// TIA Portal V16 export
// export: Created 2021-04-11T09:51:25.0986583Z, ExportSetting WithDefaults, DisplayName Totally Integrated Automation Portal, DisplayVersion V16, DisplayName TIA Portal Version Control Interface, DisplayVersion V16, DisplayName TIA Portal Openness, DisplayVersion V16, DisplayName STEP 7 Professional, DisplayVersion V16, DisplayName STEP 7 Safety, DisplayVersion V16, DisplayName WinCC Unified SCADA Engineering System, DisplayVersion V16
FUNCTION "preWorkBlock" : Void   // FC9, LAD
TITLE = Блок предработы
{ S7_Optimized_Access := 'TRUE' }
VERSION : 0.1
// Блок в котором организована работа цепей управления, аварийного останова и режимов работы
// stored: AutoNumber false, IsIECCheckEnabled false, SetENOAutomatically false, UDAEnableTagReadback false
BEGIN

REGION Network 1: удержание кнопки включение цепей управления
   // если аварийная кнопка не нажата то держим 2 секунды и цепи управления включаются
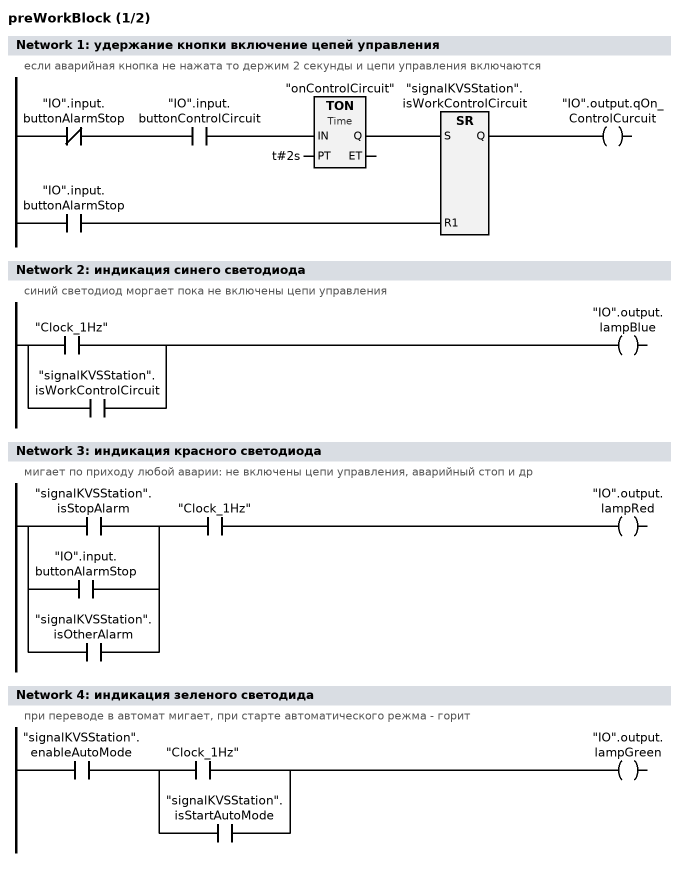
   RUNG wire#powerrail
      I_Contact( "IO".input.buttonAlarmStop )
      Contact( "IO".input.buttonControlCircuit )
      { S7_Templates := "time_type := Time" } "onControlCircuit".TON(pt := t#2s, et =>)
      S_SR(operand := "signalKVSStation".isWorkControlCircuit, r1 := wire#w1)
      Coil( "IO".output.qOn_ControlCurcuit )
   END_RUNG
   RUNG wire#powerrail
      Contact( "IO".input.buttonAlarmStop )
   END_RUNG wire#w1
   // the same network as SCL:
   "onControlCircuit".TON(IN := NOT "IO".input.buttonAlarmStop AND "IO".input.buttonControlCircuit, PT := t#2s);
   IF "onControlCircuit".Q THEN
       "signalKVSStation".isWorkControlCircuit := TRUE;   // SR flip-flop
   END_IF;
   IF "IO".input.buttonAlarmStop THEN "signalKVSStation".isWorkControlCircuit := FALSE; END_IF;
   "IO".output.qOn_ControlCurcuit := "signalKVSStation".isWorkControlCircuit;
END_REGION

REGION Network 2: индикация синего светодиода
   // синий светодиод моргает пока не включены цепи управления
   RUNG wire#powerrail
      Contact( "Clock_1Hz" )
      wire#w1
      Coil( "IO".output.lampBlue )
   END_RUNG
   RUNG wire#powerrail
      Contact( "signalKVSStation".isWorkControlCircuit )
   END_RUNG wire#w1
   // the same network as SCL:
   "IO".output.lampBlue := "Clock_1Hz" OR "signalKVSStation".isWorkControlCircuit;
END_REGION

REGION Network 3: индикация красного светодиода
   // мигает по приходу любой аварии: не включены цепи управления, аварийный стоп и др
   RUNG wire#powerrail
      Contact( "signalKVSStation".isStopAlarm )
      wire#w1
      Contact( "Clock_1Hz" )
      Coil( "IO".output.lampRed )
   END_RUNG
   RUNG wire#powerrail
      Contact( "IO".input.buttonAlarmStop )
   END_RUNG wire#w1
   RUNG wire#powerrail
      Contact( "signalKVSStation".isOtherAlarm )
   END_RUNG wire#w1
   // the same network as SCL:
   "IO".output.lampRed := ("signalKVSStation".isStopAlarm OR "IO".input.buttonAlarmStop OR "signalKVSStation".isOtherAlarm) AND "Clock_1Hz";
END_REGION

REGION Network 4: индикация зеленого светодида
   // при переводе в автомат мигает, при старте автоматического режма - горит
   RUNG wire#powerrail
      Contact( "signalKVSStation".enableAutoMode )
      wire#w1
      Contact( "Clock_1Hz" )
      wire#w2
      Coil( "IO".output.lampGreen )
   END_RUNG
   RUNG wire#w1
      Contact( "signalKVSStation".isStartAutoMode )
   END_RUNG wire#w2
   // the same network as SCL:
   "IO".output.lampGreen := "signalKVSStation".enableAutoMode AND ("Clock_1Hz" OR "signalKVSStation".isStartAutoMode);
END_REGION

REGION Network 5: разрешение на перевод в автоматический режим
   // при отсутствии аварий и нажатии кнопки автотоматического режима на панели. Данный сигнал используется как обратная связь по автоматическому и ручному режиму
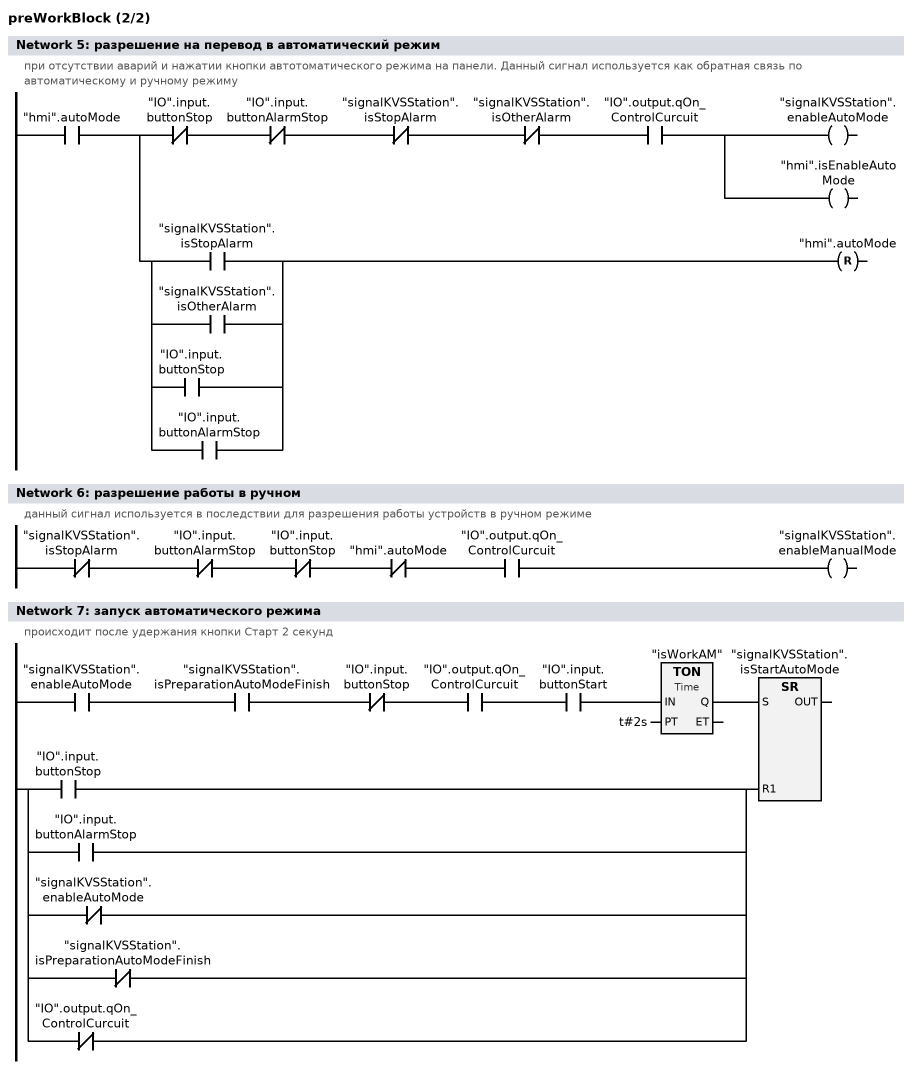
   RUNG wire#powerrail
      Contact( "hmi".autoMode )
      wire#w1
      I_Contact( "IO".input.buttonStop )
      I_Contact( "IO".input.buttonAlarmStop )
      I_Contact( "signalKVSStation".isStopAlarm )
      I_Contact( "signalKVSStation".isOtherAlarm )
      Contact( "IO".output.qOn_ControlCurcuit )
      wire#w2
      Coil( "signalKVSStation".enableAutoMode )
   END_RUNG
   RUNG wire#w2
      Coil( "hmi".isEnableAutoMode )
   END_RUNG
   RUNG wire#w1
      Contact( "signalKVSStation".isStopAlarm )
      wire#w3
      R_Coil( "hmi".autoMode )
   END_RUNG
   RUNG wire#w1
      Contact( "signalKVSStation".isOtherAlarm )
   END_RUNG wire#w3
   RUNG wire#w1
      Contact( "IO".input.buttonStop )
   END_RUNG wire#w3
   RUNG wire#w1
      Contact( "IO".input.buttonAlarmStop )
   END_RUNG wire#w3
   // the same network as SCL:
   "signalKVSStation".enableAutoMode := "hmi".autoMode AND NOT "IO".input.buttonStop AND NOT "IO".input.buttonAlarmStop AND NOT "signalKVSStation".isStopAlarm AND NOT "signalKVSStation".isOtherAlarm AND "IO".output.qOn_ControlCurcuit;
   "hmi".isEnableAutoMode := "signalKVSStation".enableAutoMode;
   IF "hmi".autoMode AND ("signalKVSStation".isStopAlarm OR "signalKVSStation".isOtherAlarm OR "IO".input.buttonStop OR "IO".input.buttonAlarmStop) THEN
       "hmi".autoMode := FALSE;
   END_IF;
END_REGION

REGION Network 6: разрешение работы в ручном
   // данный сигнал используется в последствии для разрешения работы устройств в ручном режиме
   RUNG wire#powerrail
      I_Contact( "signalKVSStation".isStopAlarm )
      I_Contact( "IO".input.buttonAlarmStop )
      I_Contact( "IO".input.buttonStop )
      I_Contact( "hmi".autoMode )
      Contact( "IO".output.qOn_ControlCurcuit )
      Coil( "signalKVSStation".enableManualMode )
   END_RUNG
   // the same network as SCL:
   "signalKVSStation".enableManualMode := NOT "signalKVSStation".isStopAlarm AND NOT "IO".input.buttonAlarmStop AND NOT "IO".input.buttonStop AND NOT "hmi".autoMode AND "IO".output.qOn_ControlCurcuit;
END_REGION

REGION Network 7: запуск автоматического режима
   // происходит после удержания кнопки Старт 2 секунд
   RUNG wire#powerrail
      Contact( "signalKVSStation".enableAutoMode )
      Contact( "signalKVSStation".isPreparationAutoModeFinish )
      I_Contact( "IO".input.buttonStop )
      Contact( "IO".output.qOn_ControlCurcuit )
      Contact( "IO".input.buttonStart )
      { S7_Templates := "time_type := Time" } "isWorkAM".TON(pt := t#2s, et =>)
      S_SR(operand := "signalKVSStation".isStartAutoMode, r1 := wire#w1)
   END_RUNG
   RUNG wire#powerrail
      Contact( "IO".input.buttonStop )
   END_RUNG wire#w1
   RUNG wire#powerrail
      Contact( "IO".input.buttonAlarmStop )
   END_RUNG wire#w1
   RUNG wire#powerrail
      I_Contact( "signalKVSStation".enableAutoMode )
   END_RUNG wire#w1
   RUNG wire#powerrail
      I_Contact( "signalKVSStation".isPreparationAutoModeFinish )
   END_RUNG wire#w1
   RUNG wire#powerrail
      I_Contact( "IO".output.qOn_ControlCurcuit )
   END_RUNG wire#w1
   // the same network as SCL:
   "isWorkAM".TON(IN := "signalKVSStation".enableAutoMode AND "signalKVSStation".isPreparationAutoModeFinish AND NOT "IO".input.buttonStop AND "IO".output.qOn_ControlCurcuit AND "IO".input.buttonStart,
                  PT := t#2s);
   IF "isWorkAM".Q THEN
       "signalKVSStation".isStartAutoMode := TRUE;   // SR flip-flop
   END_IF;
   IF "IO".input.buttonStop OR "IO".input.buttonAlarmStop OR NOT "signalKVSStation".enableAutoMode OR NOT "signalKVSStation".isPreparationAutoModeFinish OR NOT "IO".output.qOn_ControlCurcuit THEN
       "signalKVSStation".isStartAutoMode := FALSE;
   END_IF;
END_REGION
END_FUNCTION
